{attribute 'qualified_only'}
{attribute 'strict'}
TYPE STATI:
(
	S0 := 0, S1, S2, S3, SE, SA
);
END_TYPE

(* stored: Version 1.1.0.1, ProductVersion 3.1.4024.12
   EnumerationTextList STATI: Id {fedba436-bd40-4e93-a3b7-770bf0885425} *)
